(* CoDeSys 2.3 export: FB_OPENCLOSEDOOR.EXP *)

(* POU 8_TemperatureCtrl/FB_openCloseDoor, LD *)
FUNCTION_BLOCK FB_openCloseDoor
VAR_INPUT
	openInside					:BOOL;
	closeInside					:BOOL;
	openOutside					:BOOL;
	closeInside					:BOOL;
	openCloseOutside			:BOOL;
	pressureReleased			:BOOL;
	speedOverLimit				:BOOL;
	pressureLimit					:BOOL;
	pressureOK					:BOOL;
	wheelchairInLimit				:BOOL;
	additionalStepInuse			:BOOL;
	doorCloseLimit				:BOOL;
	doorOpenLImit				:BOOL;
	emergencyReleaseUsed		:BOOL;
END_VAR
VAR_OUTPUT
	doorOpen						:BOOL;
	doorClose						:BOOL;
END_VAR
VAR
	limitsinsideOK				:BOOL;
	limitsoutsideOK				:BOOL;
	reset1							:BOOL;
	reset2							:BOOL;
	sr1								:SR;
	sr2								:SR;
	sr3								:SR;
	sr4								:SR;
	doorOpenInside				:BOOL;
	doorCloseInside				:BOOL;
	doorOpenOutside				:BOOL;
	doorCloseOutside			:BOOL;
	fb1								:FB_limitOutsideDoorCntrl;
END_VAR
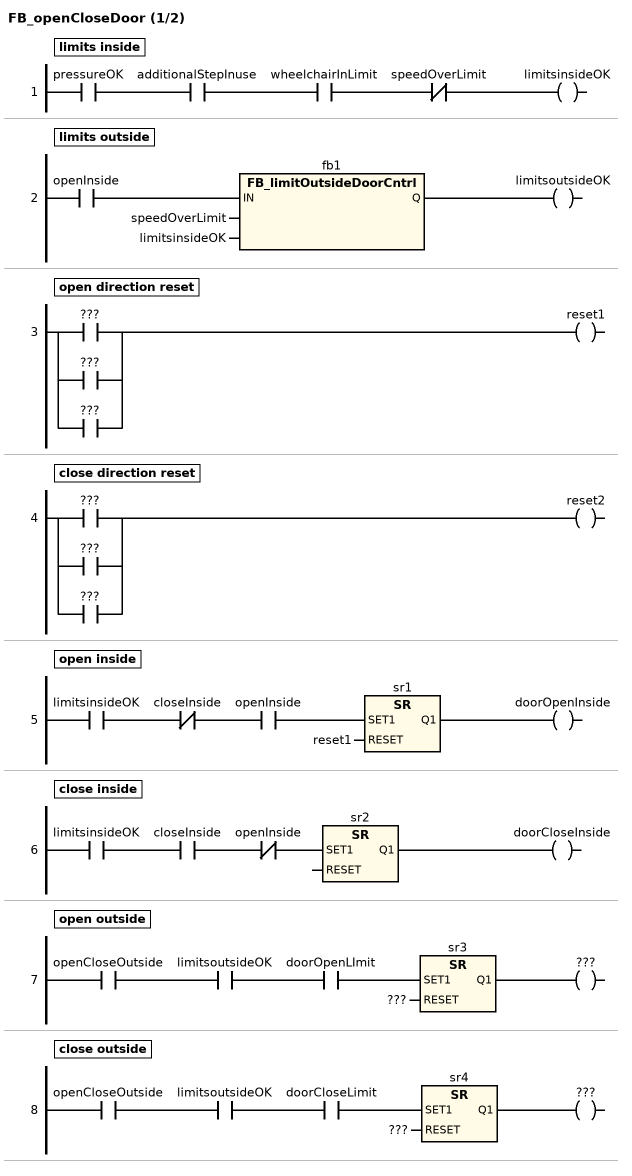
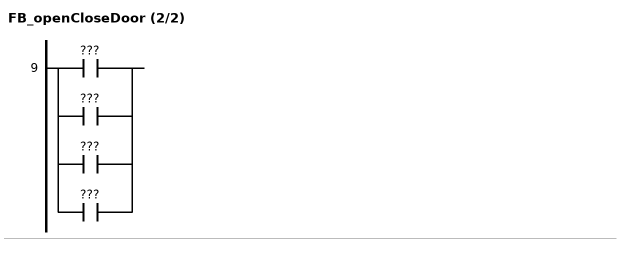
_LD_ (* Ladder Diagram *)
NETWORK 1 limits inside:
	[pressureOK] - [additionalStepInuse] - [wheelchairInLimit] - [/speedOverLimit] --- (limitsinsideOK)
NETWORK 2 limits outside:
	[openInside] - fb1:FB_limitOutsideDoorCntrl(*, speedOverLimit, limitsinsideOK) --- (limitsoutsideOK)
NETWORK 3 open direction reset:
	{ [???] | [???] | [???] } --- (reset1)
NETWORK 4 close direction reset:
	{ [???] | [???] | [???] } --- (reset2)
NETWORK 5 open inside:
	[limitsinsideOK] - [/closeInside] - [openInside] - sr1:SR(SET1: *, RESET: reset1) --- (doorOpenInside)
NETWORK 6 close inside:
	[limitsinsideOK] - [closeInside] - [/openInside] - sr2:SR(SET1: *, RESET: ) --- (doorCloseInside)
NETWORK 7 open outside:
	[openCloseOutside] - [limitsoutsideOK] - [doorOpenLImit] - sr3:SR(SET1: *, RESET: ???) --- (???)
NETWORK 8 close outside:
	[openCloseOutside] - [limitsoutsideOK] - [doorCloseLimit] - sr4:SR(SET1: *, RESET: ???) --- (???)
NETWORK 9
	{ [???] | [???] | [???] | [???] }
_END_LD_
(* the same logic as Structured Text *)
(* Network 1 *)
limitsinsideOK := pressureOK AND additionalStepInuse AND wheelchairInLimit AND NOT speedOverLimit;
(* Network 2: see the listing above *)
(* Network 3: see the listing above *)
(* Network 4: see the listing above *)
(* Network 5 *)
sr1(SET1 := limitsinsideOK AND NOT closeInside AND openInside, RESET := reset1);
doorOpenInside := sr1.Q1;
(* Network 6: see the listing above *)
(* Network 7: see the listing above *)
(* Network 8: see the listing above *)
(* Network 9: see the listing above *)
END_FUNCTION_BLOCK
